Staubli VAL3: FILEDIR.dtx

mdesc mNomSpeed
num nFile2ID
num nFileID
string sBuff
